INTERFACE I_Collectable EXTENDS __SYSTEM.IQueryInterface

END_INTERFACE

(* stored: Version 1.1.0.1, ProductVersion 3.1.4024.11
   Itf I_Collectable: Id {91963344-e17c-413b-a406-3e7ed7a0798a} *)
